TYPE (* IEC61131-3, Table 14#5 *)
  (* Standard: 1131-3 *)
  (* Version 0.0, 10/1/2026, Schneider Electric, Template *)
  PACKAGE Main;
  {SET_ATTRIBUTE(nxtDataType, R/SPXHgkKnU1woEFbZXR/WE9SnZiyLHfnNZtF7UdWdlOgcpfNFTOwqc6FhIuGnWoJ2qqfcE/unnJds7ZkdI9kg==)}
  dtEnum : USINT (
    Stop := 0,
    Run := 1,
    Fault := 2
  );
END_TYPE
